TYPE typeSeqRow :
STRUCT
	Advance:typeAutoRowMotion;
	Returnn:typeAutoRowMotion; //return is a keyword now?
END_STRUCT
END_TYPE

(* stored: Version 1.1.0.1, ProductVersion 3.1.4024.11
   DUT typeSeqRow: Id {7140d2f4-c7a6-001c-23c6-e26698270501} *)
